FUNCTION_BLOCK EL2088
VAR
	{attribute addProperty Name "WcState"}
	_wcState : WcStateBase;
	{attribute addProperty Name "Info data"}
	_infoData : InfoDataBase;
	_io : EL2xx8_Data;
END_VAR

PROPERTY IO : REFERENCE TO EL2xx8_Data
GET
IO REF= _io;
END_GET
END_PROPERTY

PROPERTY WcState : REFERENCE TO WcStateBase
GET
WcState REF= _wcState;
END_GET
END_PROPERTY

END_FUNCTION_BLOCK

(* stored: Version 1.1.0.1, ProductVersion 3.1.4024.9
   POU EL2088: Id {73c94b27-5a8f-0410-1c8a-f62b4b400d51}, SpecialFunc None
   Property IO: Id {c1a5eefe-35c7-0fc4-2e70-98578311114d}
   Get Get: Id {df2eb7e2-a738-0389-35c0-973ce6a00972}
   Property WcState: Id {511c10e2-114a-0791-2e72-fe062611a39f}
   Get Get: Id {93ad00b2-0282-0125-115a-257cc4cc4edc} *)
